Omron Sysmac Studio project Production_Rate_Calculator (Sysmac Studio 1.64.0.64008, StandardProject)

# Controller new_Controller_0: NX1P2-9024DT1 version 1.69
Units and slaves: Unit 1 : NX-PF0730 (N1); Unit 2 : NX-ID4442 (N2); Unit 3 : NX-OD4256 (N3)
Task PrimaryTask (priority 4, period or condition 2000): line_1

PROGRAM line_1
VAR
    machine_1_prodection_rate : FB_ProductionRateMonitor;
    i_tb_sensor : BOOL;
    i_reser_button : BOOL;
    avrage_time : TIME;
    part_in_minut : LREAL;
END_VAR
machine_1_prodection_rate(i_ProductPresenceSensor:=i_tb_sensor,
		i_TargetProductionQuantity:=10,
		i_ResetProductionMeasurement:= i_reser_button,
		t_AverageCycleTimePerPart => avrage_time,
		o_PartPerMinut=>part_in_minut);
END_PROGRAM

FUNCTION_BLOCK FB_ProductionRateMonitor
VAR
    fb_ProductDetectionEdge : R_TRIG;
    ProducedPartCount : INT;
    x_CycleTimeMeasurementActive : bool;
    fb_ProductionElapsedTimer : TON;
    t_ProductionElapsedTime : TIME;
    t_TotalProductionTime : TIME;
    li_TotalProductionTimeNs : LINT;
    li_AverageCycleTimeNs : LINT;
END_VAR
VAR_INPUT
    i_ProductPresenceSensor : BOOL;
    i_TargetProductionQuantity : int;
    i_ResetProductionMeasurement : bool;
END_VAR
VAR_OUTPUT
    t_AverageCycleTimePerPart : time;
    o_PartPerMinut : LREAL;
END_VAR
//==============================================================
// PRODUCTION RATE MONITOR
//==============================================================


//--------------------------------------------------------------
// Rising Edge Detection for Product Presence Sensor
//--------------------------------------------------------------
fb_ProductDetectionEdge(
    CLK := i_ProductPresenceSensor
);


//--------------------------------------------------------------
// Count Produced Parts Until Target Production Quantity
// Is Reached
//--------------------------------------------------------------
IF fb_ProductDetectionEdge.Q AND
   NOT (ProducedPartCount >= i_TargetProductionQuantity) THEN

    x_CycleTimeMeasurementActive := TRUE;
    ProducedPartCount := ProducedPartCount + 1;

END_IF;


//--------------------------------------------------------------
// Production Elapsed Time Measurement
//--------------------------------------------------------------
fb_ProductionElapsedTimer(
    IN := x_CycleTimeMeasurementActive,
    PT := T#90s,
    ET => t_ProductionElapsedTime
);


//--------------------------------------------------------------
// Update Production Time and Calculate Production Rate
//--------------------------------------------------------------
IF x_CycleTimeMeasurementActive THEN

    // Update total production time
    t_TotalProductionTime := t_ProductionElapsedTime;


    // Convert production time from TIME to nanoseconds
    li_TotalProductionTimeNs :=
        TimeToNanoSec(
            In := t_TotalProductionTime
        );


    //----------------------------------------------------------
    // Calculate Average Cycle Time Per Part
    //----------------------------------------------------------
    IF ProducedPartCount > 0 THEN

        li_AverageCycleTimeNs :=
            li_TotalProductionTimeNs / ProducedPartCount;


        //------------------------------------------------------
        // Calculate Production Rate in Parts Per Minute
        //------------------------------------------------------
        IF li_TotalProductionTimeNs > 0 THEN

            o_PartPerMinut :=
                INT_TO_LREAL(ProducedPartCount) *
                60000000000.0 /
                LINT_TO_LREAL(li_TotalProductionTimeNs);

        END_IF;

    END_IF;

END_IF;


//--------------------------------------------------------------
// Stop Cycle Time Measurement After Target Quantity Is Reached
//--------------------------------------------------------------
IF ProducedPartCount >= i_TargetProductionQuantity THEN

    x_CycleTimeMeasurementActive := FALSE;

END_IF;


//--------------------------------------------------------------
// Reset Production Measurement
//--------------------------------------------------------------
IF i_ResetProductionMeasurement THEN

    ProducedPartCount := 0;

    li_TotalProductionTimeNs := 0;

    li_AverageCycleTimeNs := 0;

    t_TotalProductionTime := T#0s;

    t_AverageCycleTimePerPart := T#0s;

    o_PartPerMinut := 0.0;

END_IF;


//--------------------------------------------------------------
// Convert Average Cycle Time from Nanoseconds to TIME
//--------------------------------------------------------------
t_AverageCycleTimePerPart :=
    NanoSecToTime(
        In := li_AverageCycleTimeNs
    );
END_FUNCTION_BLOCK